(* IEC 61131-3 sources: Industry-PLC-LLM/data/PLCBEAD_repo/PLCBEAD_PLCEmbed-main/PLC-BEAD/Source/GEB/R2_DIV, 1 file *)

(* ---- R2_DIV.ST ---- *)
TYPE REAL2 :

	STRUCT
		R1  : REAL;
		RX : REAL;
	END_STRUCT;

END_TYPE

FUNCTION_BLOCK R2_DIV_Block

	VAR_INPUT
		X :	REAL2;
		Y :	REAL;
	END_VAR

	VAR_OUTPUT
		R2_DIV :	REAL2;
	END_VAR

	R2_DIV.RX := X.RX / Y;
	R2_DIV.R1  := X.R1  / Y;

END_FUNCTION_BLOCK

PROGRAM program0

	VAR
		X :	REAL2;
		Y :	REAL;

        R2_DIV :	REAL2;
		func_block : R2_DIV_Block;
	END_VAR
	func_block.X := X;
	func_block.Y := Y;
	func_block();
	R2_DIV := func_block.R2_DIV;

END_PROGRAM
